FUNCTION_BLOCK EA_2_router
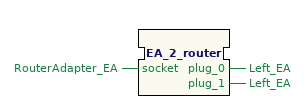
  SOCKETS
    socket : RouterAdapter_EA;
  END_SOCKETS
  PLUGS
    plug_0 : Left_EA;
    plug_1 : Left_EA;
  END_PLUGS
  FBS
    EA_2_leftSwitch : EA_2_leftSwitch;
    EA_2_rightSwitch : EA_2_rightSwitch;
  END_FBS
  EVENT_CONNECTIONS
    socket.O_event1 TO EA_2_leftSwitch.O_event1;
    socket.O_event2 TO EA_2_leftSwitch.O_event2;
    socket.S_O_Event1 TO EA_2_leftSwitch.S_O_Event1;
    socket.S_O_Event2 TO EA_2_leftSwitch.S_O_Event2;
    EA_2_leftSwitch.O_event1_0 TO plug_0.O_event1;
    EA_2_leftSwitch.O_event2_0 TO plug_0.O_event2;
    EA_2_leftSwitch.S_O_Event1_0 TO plug_0.S_O_Event1;
    EA_2_leftSwitch.S_O_Event2_0 TO plug_0.S_O_Event2;
    EA_2_leftSwitch.O_event1_1 TO plug_1.O_event1;
    EA_2_leftSwitch.O_event2_1 TO plug_1.O_event2;
    EA_2_leftSwitch.S_O_Event1_1 TO plug_1.S_O_Event1;
    EA_2_leftSwitch.S_O_Event2_1 TO plug_1.S_O_Event2;
    EA_2_rightSwitch.I_event1 TO socket.I_event1;
    EA_2_rightSwitch.I_event2 TO socket.I_event2;
    EA_2_rightSwitch.S_I_Event1 TO socket.S_I_Event1;
    EA_2_rightSwitch.S_I_Event2 TO socket.S_I_Event2;
    plug_0.I_event1 TO EA_2_rightSwitch.I_event1_0;
    plug_0.I_event2 TO EA_2_rightSwitch.I_event2_0;
    plug_0.S_I_Event1 TO EA_2_rightSwitch.S_I_Event1_0;
    plug_0.S_I_Event2 TO EA_2_rightSwitch.S_I_Event2_0;
    plug_1.I_event1 TO EA_2_rightSwitch.I_event1_1;
    plug_1.I_event2 TO EA_2_rightSwitch.I_event2_1;
    plug_1.S_I_Event1 TO EA_2_rightSwitch.S_I_Event1_1;
    plug_1.S_I_Event2 TO EA_2_rightSwitch.S_I_Event2_1;
  END_CONNECTIONS
  DATA_CONNECTIONS
    socket.O_data1 TO EA_2_leftSwitch.O_data1;
    socket.O_data2 TO EA_2_leftSwitch.O_data2;
    socket.S_O_data1 TO EA_2_leftSwitch.S_O_data1;
    socket.S_O_data2 TO EA_2_leftSwitch.S_O_data2;
    socket.O_router TO EA_2_leftSwitch.O_router;
    EA_2_leftSwitch.O_data1_0 TO plug_0.O_data1;
    EA_2_leftSwitch.O_data2_0 TO plug_0.O_data2;
    EA_2_leftSwitch.S_O_data1_0 TO plug_0.S_O_data1;
    EA_2_leftSwitch.S_O_data2_0 TO plug_0.S_O_data2;
    EA_2_leftSwitch.O_data1_1 TO plug_1.O_data1;
    EA_2_leftSwitch.O_data2_1 TO plug_1.O_data2;
    EA_2_leftSwitch.S_O_data1_1 TO plug_1.S_O_data1;
    EA_2_leftSwitch.S_O_data2_1 TO plug_1.S_O_data2;
    EA_2_rightSwitch.I_data1 TO socket.I_data1;
    EA_2_rightSwitch.I_data2 TO socket.I_data2;
    EA_2_rightSwitch.S_I_data1 TO socket.S_I_data1;
    EA_2_rightSwitch.S_I_data2 TO socket.S_I_data2;
    EA_2_rightSwitch.I_router TO socket.I_router;
    plug_0.I_data1 TO EA_2_rightSwitch.I_data1_0;
    plug_0.I_data2 TO EA_2_rightSwitch.I_data2_0;
    plug_0.S_I_data1 TO EA_2_rightSwitch.S_I_data1_0;
    plug_0.S_I_data2 TO EA_2_rightSwitch.S_I_data2_0;
    plug_1.I_data1 TO EA_2_rightSwitch.I_data1_1;
    plug_1.I_data2 TO EA_2_rightSwitch.I_data2_1;
    plug_1.S_I_data1 TO EA_2_rightSwitch.S_I_data1_1;
    plug_1.S_I_data2 TO EA_2_rightSwitch.S_I_data2_1;
  END_CONNECTIONS
END_FUNCTION_BLOCK
